INTERFACE I_EnumeratorParent

METHOD RemoveEnumerator
VAR_INPUT
	Enumerator : I_Enumerator;
END_VAR
END_METHOD

END_INTERFACE

(* stored: Version 1.1.0.1, ProductVersion 3.1.4024.12
   Itf I_EnumeratorParent: Id {a33e7360-a393-43a1-974e-8deab5aa505c}
   Method RemoveEnumerator: Id {4b8e8e66-95f0-4c2f-ba75-df776b57149d} *)
